TYPE Machine_Info :
STRUCT
	Machine_Serial_Number : STRING;
	Electrical_Bill_ID : STRING;
	Purchase_Order_Number : STRING;
	Work_Order_Number : STRING;
END_STRUCT
END_TYPE

(* stored: Version 1.1.0.1, ProductVersion 3.1.4024.12
   DUT Machine_Info: Id {9c1150c1-8f25-4e7e-bc17-a2a1b6ebb7d8} *)
